{attribute addProperty BoxType "AT2026-0250-0022"}
{attribute addProperty Id "A_0079_AT2002_5249_0018_AT2002_5249AT2002_C5E5984862678.25"}
{attribute addProperty CRC "3492801648"}
{attribute addProperty SizeInBites "626"}
{attribute addProperty SizeInBytes "78.25"}
TYPE A_0067_AT2026_0250_0022_AT2026_0250_D02FEC70 EXTENDS AT2026_BA5A9548 :
STRUCT
	{attribute addProperty Name "A_0079_AT2002_5249_0018_AT2002_5249"}
	A_0079_AT2002_5249_0018_AT2002_5249 : AT2002_C5E59848;
END_STRUCT
END_TYPE

(* stored: Version 1.2.0.0, ProductVersion 3.1.4024.9
   DUT A_0067_AT2026_0250_0022_AT2026_0250_D02FEC70: Id {1f20f4b3-26b0-4561-ab41-a5f7d291b169} *)
